// TIA Portal V16 export
// export: Created 2020-12-17T10:43:18.8581379Z, ExportSetting WithDefaults, WithReadOnly, DisplayName Totally Integrated Automation Portal, DisplayVersion V16 Update 2, DisplayName TIA Portal Version Control Interface, DisplayVersion V16 Update 2, DisplayName TIA Portal Openness, DisplayVersion V16 Update 2, DisplayName STEP 7 Professional, DisplayVersion V16 Update 2, DisplayName STEP 7 Safety, DisplayVersion V16, DisplayName WinCC Advanced / Unified PC, DisplayVersion V16 Update 2
DATA_BLOCK "Data_block_2"   // DB3
{ S7_Optimized_Access := 'TRUE' }
VERSION : 0.1
// stored: AutoNumber true, CodeModifiedDate 2020-12-17T10:42:33.3081896Z, CompileDate 2020-12-17T10:42:38.4660302Z, CreationDate 2020-12-17T10:42:13.2923269Z, DBAccessibleFromOPCUA true, DownloadWithoutReinit false, InterfaceModifiedDate 2020-12-17T10:42:33.3081896Z, IsConsistent true, IsKnowHowProtected false, IsOnlyStoredInLoadMemory false, IsPLCDB false, IsRetainMemResEnabled false, IsWriteProtectedInAS false, MemoryReserve 100, ModifiedDate 2020-12-17T10:42:33.3081896Z, ParameterModified 2020-12-17T10:42:33.3081896Z, StructureModified 2020-12-17T10:42:33.3081896Z
   VAR
      p1 { S7_SetPoint := 'True'} : "Point";
   END_VAR
   VAR RETAIN
      p2 { S7_SetPoint := 'True'} : "Point";
   END_VAR
   VAR
      p3 { S7_SetPoint := 'True'} : "Point";
   END_VAR
   VAR RETAIN
      p4 { S7_SetPoint := 'True'} : "Point";
   END_VAR
BEGIN
END_DATA_BLOCK
